Xinje XDPPro project, PLC1: XD5E-60 (software 3.8.0a 2025-04-30)

PROGRAM 梯形图

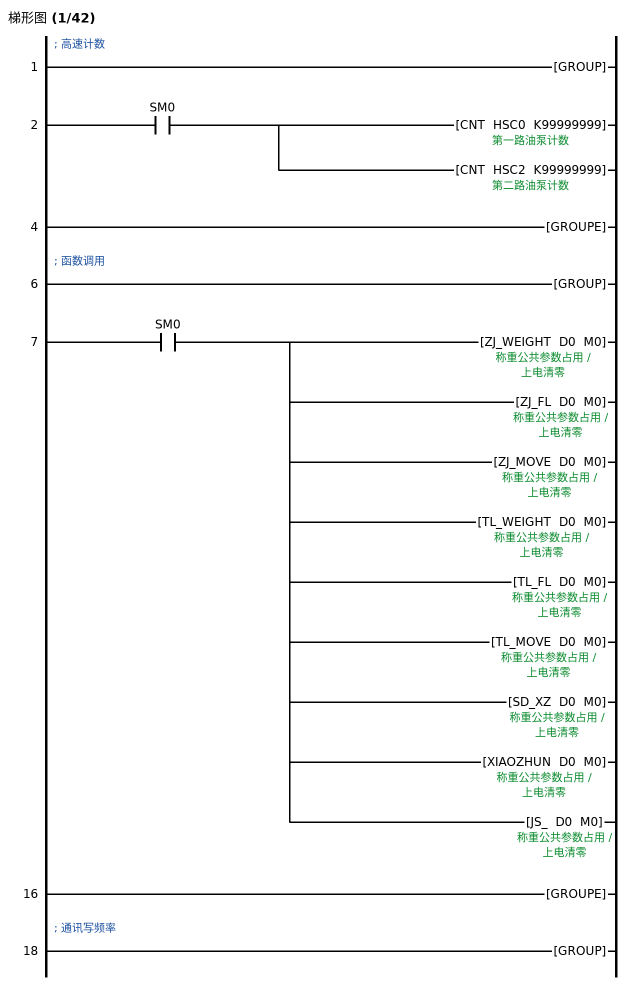
; 高速计数
GROUP
LD     SM0
CNT    HSC0 K99999999	; 第一路油泵计数
CNT    HSC2 K99999999	; 第二路油泵计数
GROUPE
; 函数调用
GROUP
LD     SM0
ZJ_WEIGHT D0 M0	; 称重公共参数占用 / 上电清零
ZJ_FL  D0 M0	; 称重公共参数占用 / 上电清零
ZJ_MOVE D0 M0	; 称重公共参数占用 / 上电清零
TL_WEIGHT D0 M0	; 称重公共参数占用 / 上电清零
TL_FL  D0 M0	; 称重公共参数占用 / 上电清零
TL_MOVE D0 M0	; 称重公共参数占用 / 上电清零
SD_XZ  D0 M0	; 称重公共参数占用 / 上电清零
XIAOZHUN D0 M0	; 称重公共参数占用 / 上电清零
JS_    D0 M0	; 称重公共参数占用 / 上电清零
GROUPE
; 通讯写频率
GROUP

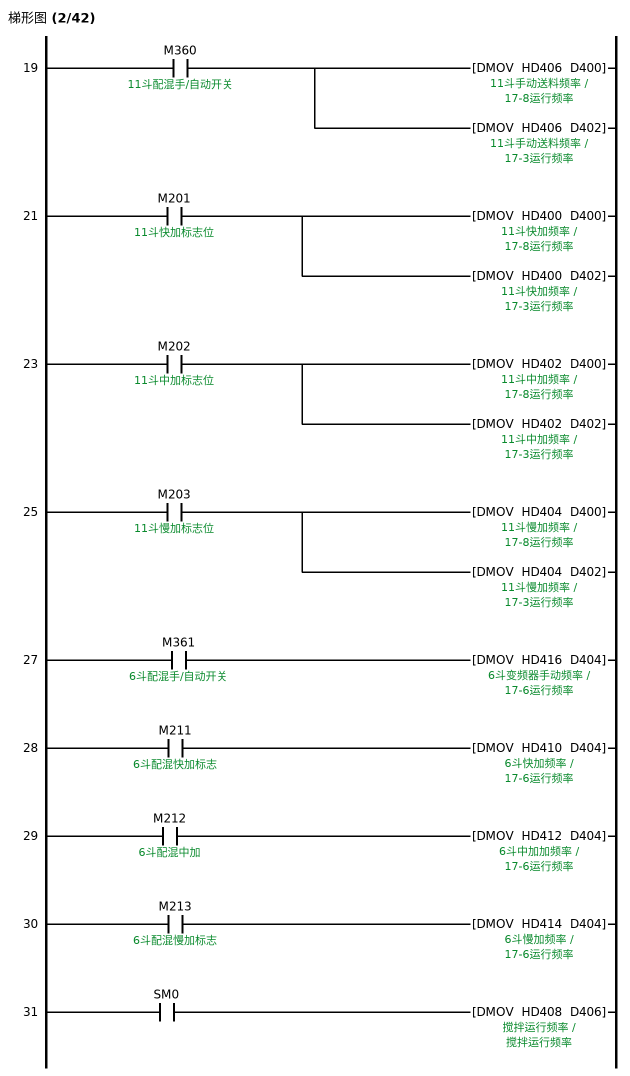
LD     M360	; 11斗配混手/自动开关
DMOV   HD406 D400	; 11斗手动送料频率 / 17-8运行频率
DMOV   HD406 D402	; 11斗手动送料频率 / 17-3运行频率
LD     M201	; 11斗快加标志位
DMOV   HD400 D400	; 11斗快加频率 / 17-8运行频率
DMOV   HD400 D402	; 11斗快加频率 / 17-3运行频率
LD     M202	; 11斗中加标志位
DMOV   HD402 D400	; 11斗中加频率 / 17-8运行频率
DMOV   HD402 D402	; 11斗中加频率 / 17-3运行频率
LD     M203	; 11斗慢加标志位
DMOV   HD404 D400	; 11斗慢加频率 / 17-8运行频率
DMOV   HD404 D402	; 11斗慢加频率 / 17-3运行频率
LD     M361	; 6斗配混手/自动开关
DMOV   HD416 D404	; 6斗变频器手动频率 / 17-6运行频率
LD     M211	; 6斗配混快加标志
DMOV   HD410 D404	; 6斗快加频率 / 17-6运行频率
LD     M212	; 6斗配混中加
DMOV   HD412 D404	; 6斗中加加频率 / 17-6运行频率
LD     M213	; 6斗配混慢加标志
DMOV   HD414 D404	; 6斗慢加频率 / 17-6运行频率
LD     SM0
DMOV   HD408 D406	; 搅拌运行频率 / 搅拌运行频率

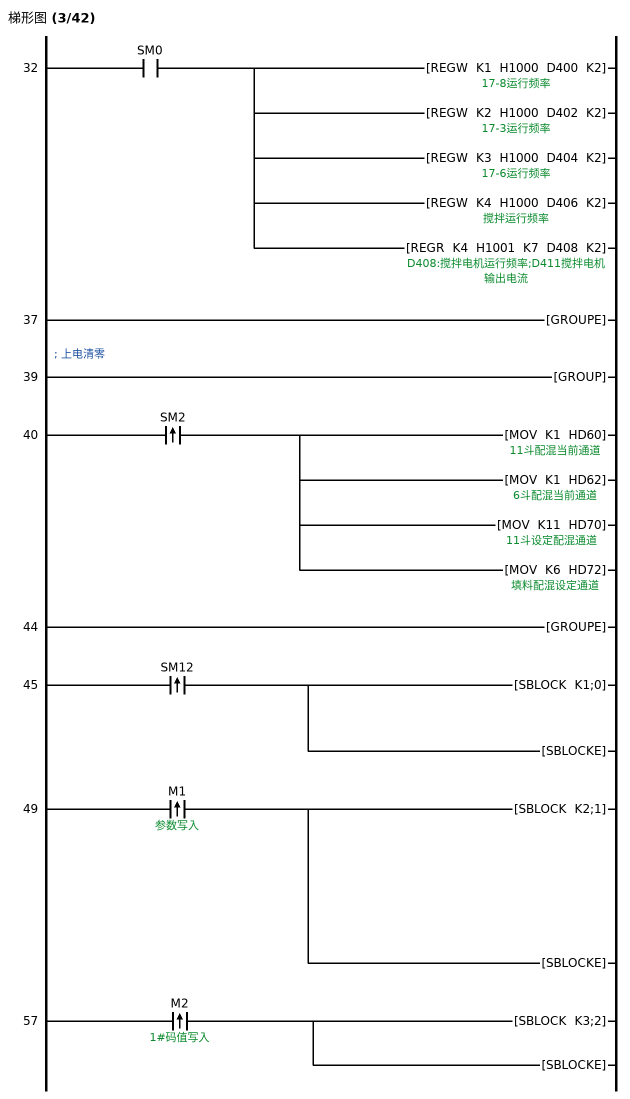
LD     SM0
REGW   K1 H1000 D400 K2	; 17-8运行频率
REGW   K2 H1000 D402 K2	; 17-3运行频率
REGW   K3 H1000 D404 K2	; 17-6运行频率
REGW   K4 H1000 D406 K2	; 搅拌运行频率
REGR   K4 H1001 K7 D408 K2	; D408:搅拌电机运行频率;D411搅拌电机输出电流
GROUPE
; 上电清零
GROUP
LDP    SM2
MOV    K1 HD60	; 11斗配混当前通道
MOV    K1 HD62	; 6斗配混当前通道
MOV    K11 HD70	; 11斗设定配混通道
MOV    K6 HD72	; 填料配混设定通道
GROUPE
LDP    SM12
SBLOCK K1;0
SBLOCKE
LDP    M1	; 参数写入
SBLOCK K2;1
SBLOCKE
LDP    M2	; 1#码值写入
SBLOCK K3;2
SBLOCKE

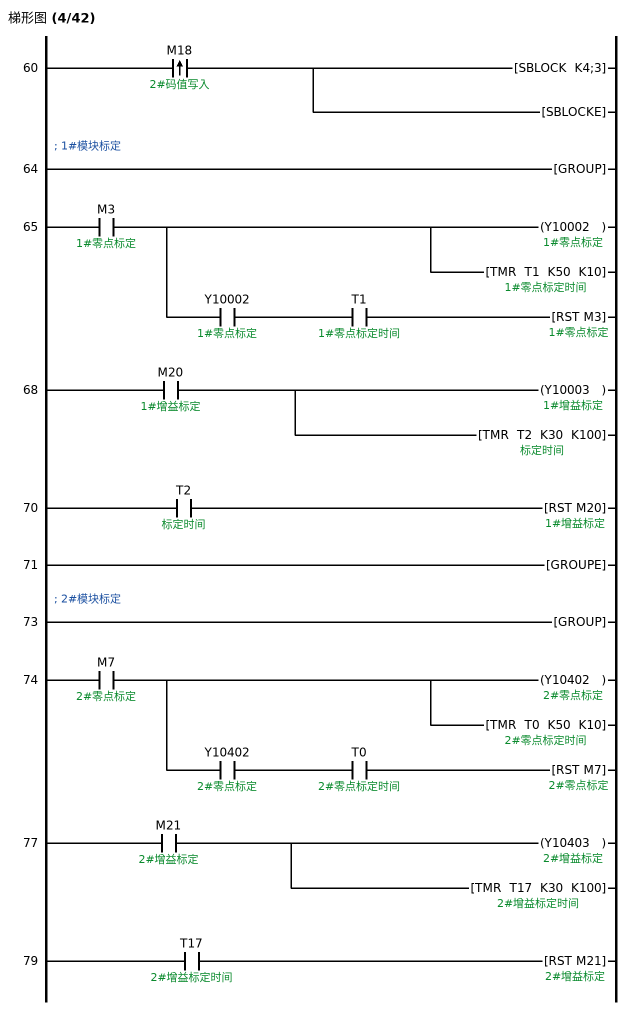
LDP    M18	; 2#码值写入
SBLOCK K4;3
SBLOCKE
; 1#模块标定
GROUP
LD     M3	; 1#零点标定
OUT    Y10002	; 1#零点标定
TMR    T1 K50 K10	; 1#零点标定时间
AND    Y10002	; 1#零点标定
AND    T1	; 1#零点标定时间
RST    M3	; 1#零点标定
LD     M20	; 1#增益标定
OUT    Y10003	; 1#增益标定
TMR    T2 K30 K100	; 标定时间
LD     T2	; 标定时间
RST    M20	; 1#增益标定
GROUPE
; 2#模块标定
GROUP
LD     M7	; 2#零点标定
OUT    Y10402	; 2#零点标定
TMR    T0 K50 K10	; 2#零点标定时间
AND    Y10402	; 2#零点标定
AND    T0	; 2#零点标定时间
RST    M7	; 2#零点标定
LD     M21	; 2#增益标定
OUT    Y10403	; 2#增益标定
TMR    T17 K30 K100	; 2#增益标定时间
LD     T17	; 2#增益标定时间
RST    M21	; 2#增益标定

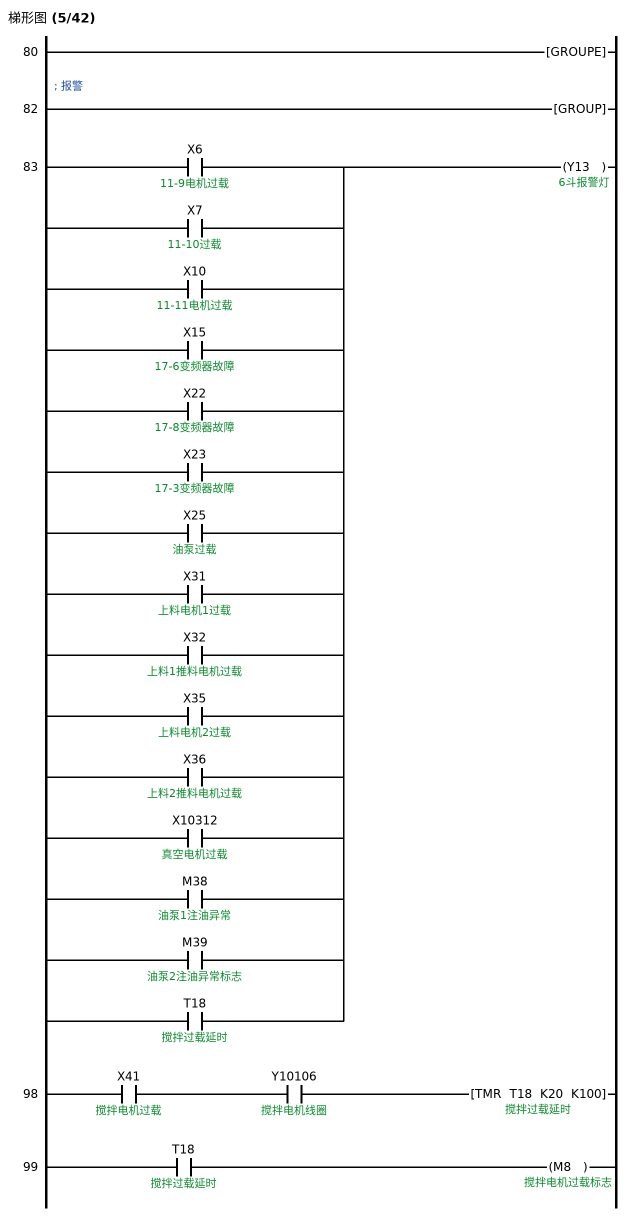
GROUPE
; 报警
GROUP
LD     X6	; 11-9电机过载
OR     X7	; 11-10过载
OR     X10	; 11-11电机过载
OR     X15	; 17-6变频器故障
OR     X22	; 17-8变频器故障
OR     X23	; 17-3变频器故障
OR     X25	; 油泵过载
OR     X31	; 上料电机1过载
OR     X32	; 上料1推料电机过载
OR     X35	; 上料电机2过载
OR     X36	; 上料2推料电机过载
OR     X10312	; 真空电机过载
OR     M38	; 油泵1注油异常
OR     M39	; 油泵2注油异常标志
OR     T18	; 搅拌过载延时
OUT    Y13	; 6斗报警灯
LD     X41	; 搅拌电机过载
AND    Y10106	; 搅拌电机线圈
TMR    T18 K20 K100	; 搅拌过载延时
LD     T18	; 搅拌过载延时
OUT    M8	; 搅拌电机过载标志

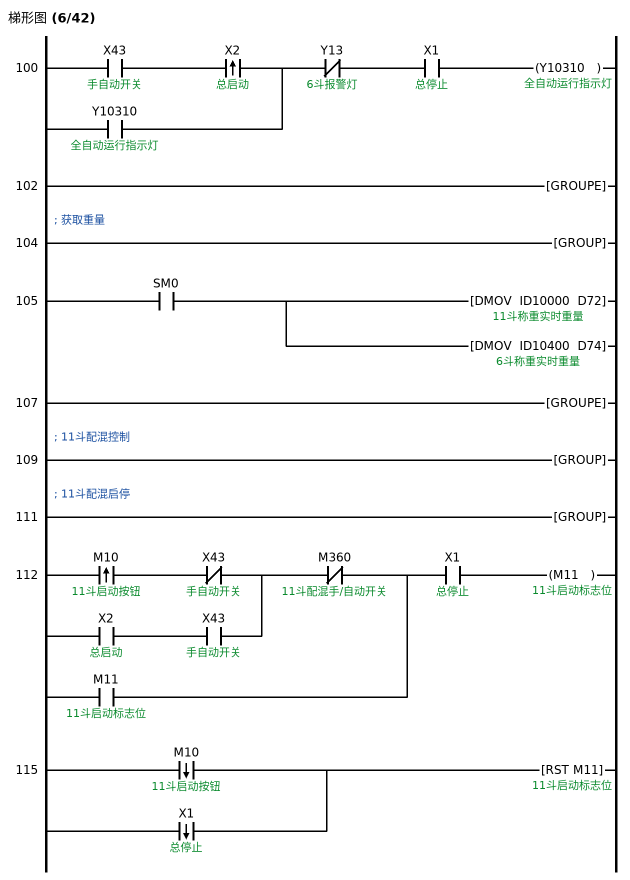
LD     X43	; 手自动开关
ANDP   X2	; 总启动
OR     Y10310	; 全自动运行指示灯
ANI    Y13	; 6斗报警灯
AND    X1	; 总停止
OUT    Y10310	; 全自动运行指示灯
GROUPE
; 获取重量
GROUP
LD     SM0
DMOV   ID10000 D72	; 11斗称重实时重量
DMOV   ID10400 D74	; 6斗称重实时重量
GROUPE
; 11斗配混控制
GROUP
; 11斗配混启停
GROUP
LDP    M10	; 11斗启动按钮
ANI    X43	; 手自动开关
LD     X2	; 总启动
AND    X43	; 手自动开关
ORB
ANI    M360	; 11斗配混手/自动开关
OR     M11	; 11斗启动标志位
AND    X1	; 总停止
OUT    M11	; 11斗启动标志位
LDF    M10	; 11斗启动按钮
ORF    X1	; 总停止
RST    M11	; 11斗启动标志位

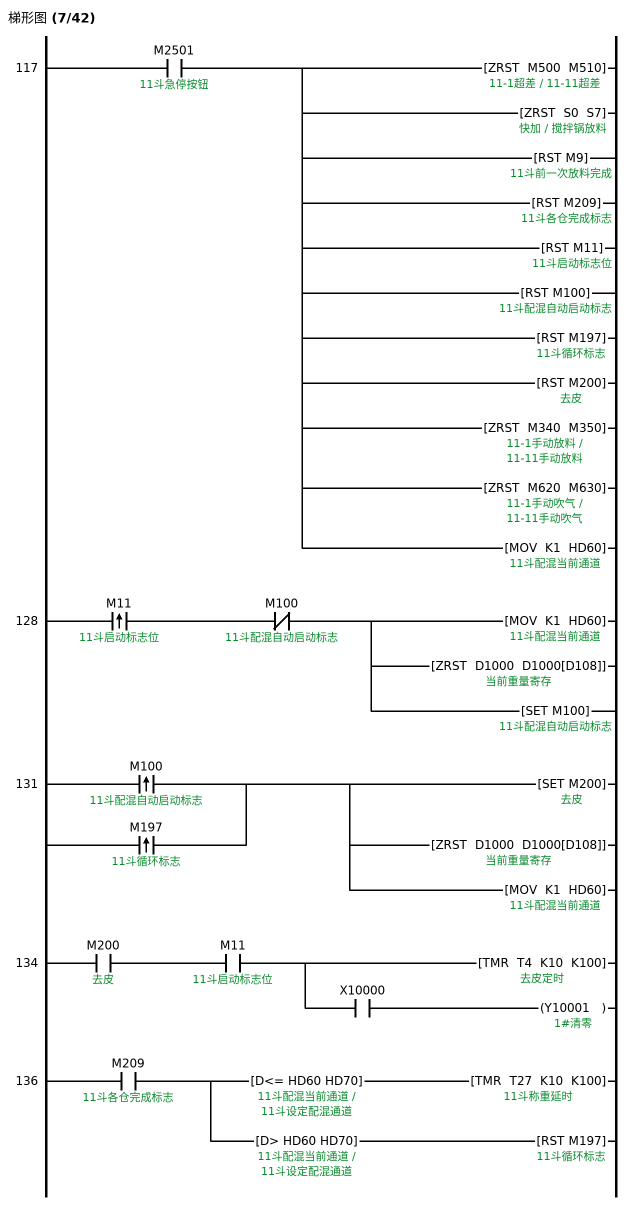
LD     M2501	; 11斗急停按钮
ZRST   M500 M510	; 11-1超差 / 11-11超差
ZRST   S0 S7	; 快加 / 搅拌锅放料
RST    M9	; 11斗前一次放料完成
RST    M209	; 11斗各仓完成标志
RST    M11	; 11斗启动标志位
RST    M100	; 11斗配混自动启动标志
RST    M197	; 11斗循环标志
RST    M200	; 去皮
ZRST   M340 M350	; 11-1手动放料 / 11-11手动放料
ZRST   M620 M630	; 11-1手动吹气 / 11-11手动吹气
MOV    K1 HD60	; 11斗配混当前通道
LDP    M11	; 11斗启动标志位
ANI    M100	; 11斗配混自动启动标志
MOV    K1 HD60	; 11斗配混当前通道
ZRST   D1000 D1000[D108]	; 当前重量寄存
SET    M100	; 11斗配混自动启动标志
LDP    M100	; 11斗配混自动启动标志
ORP    M197	; 11斗循环标志
SET    M200	; 去皮
ZRST   D1000 D1000[D108]	; 当前重量寄存
MOV    K1 HD60	; 11斗配混当前通道
LD     M200	; 去皮
AND    M11	; 11斗启动标志位
TMR    T4 K10 K100	; 去皮定时
AND    X10000
OUT    Y10001	; 1#清零
LD     M209	; 11斗各仓完成标志
MPS
DAND<= HD60 HD70	; 11斗配混当前通道 / 11斗设定配混通道
TMR    T27 K10 K100	; 11斗称重延时
MPP
DAND>  HD60 HD70	; 11斗配混当前通道 / 11斗设定配混通道
RST    M197	; 11斗循环标志

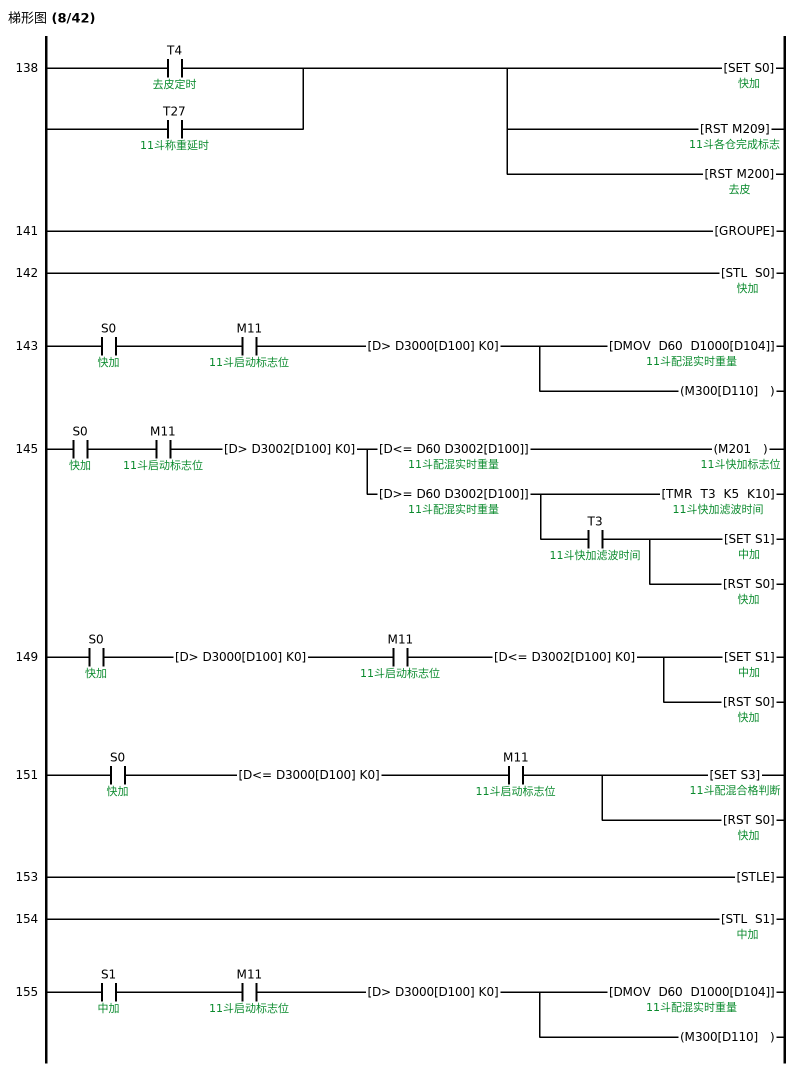
LD     T4	; 去皮定时
OR     T27	; 11斗称重延时
SET    S0	; 快加
RST    M209	; 11斗各仓完成标志
RST    M200	; 去皮
GROUPE
STL    S0	; 快加
LD     S0	; 快加
AND    M11	; 11斗启动标志位
DAND>  D3000[D100] K0
DMOV   D60 D1000[D104]	; 11斗配混实时重量
OUT    M300[D110]
LD     S0	; 快加
AND    M11	; 11斗启动标志位
DAND>  D3002[D100] K0
MPS
DAND<= D60 D3002[D100]	; 11斗配混实时重量
OUT    M201	; 11斗快加标志位
MPP
DAND>= D60 D3002[D100]	; 11斗配混实时重量
TMR    T3 K5 K10	; 11斗快加滤波时间
AND    T3	; 11斗快加滤波时间
SET    S1	; 中加
RST    S0	; 快加
LD     S0	; 快加
DAND>  D3000[D100] K0
AND    M11	; 11斗启动标志位
DAND<= D3002[D100] K0
SET    S1	; 中加
RST    S0	; 快加
LD     S0	; 快加
DAND<= D3000[D100] K0
AND    M11	; 11斗启动标志位
SET    S3	; 11斗配混合格判断
RST    S0	; 快加
STLE
STL    S1	; 中加
LD     S1	; 中加
AND    M11	; 11斗启动标志位
DAND>  D3000[D100] K0
DMOV   D60 D1000[D104]	; 11斗配混实时重量
OUT    M300[D110]

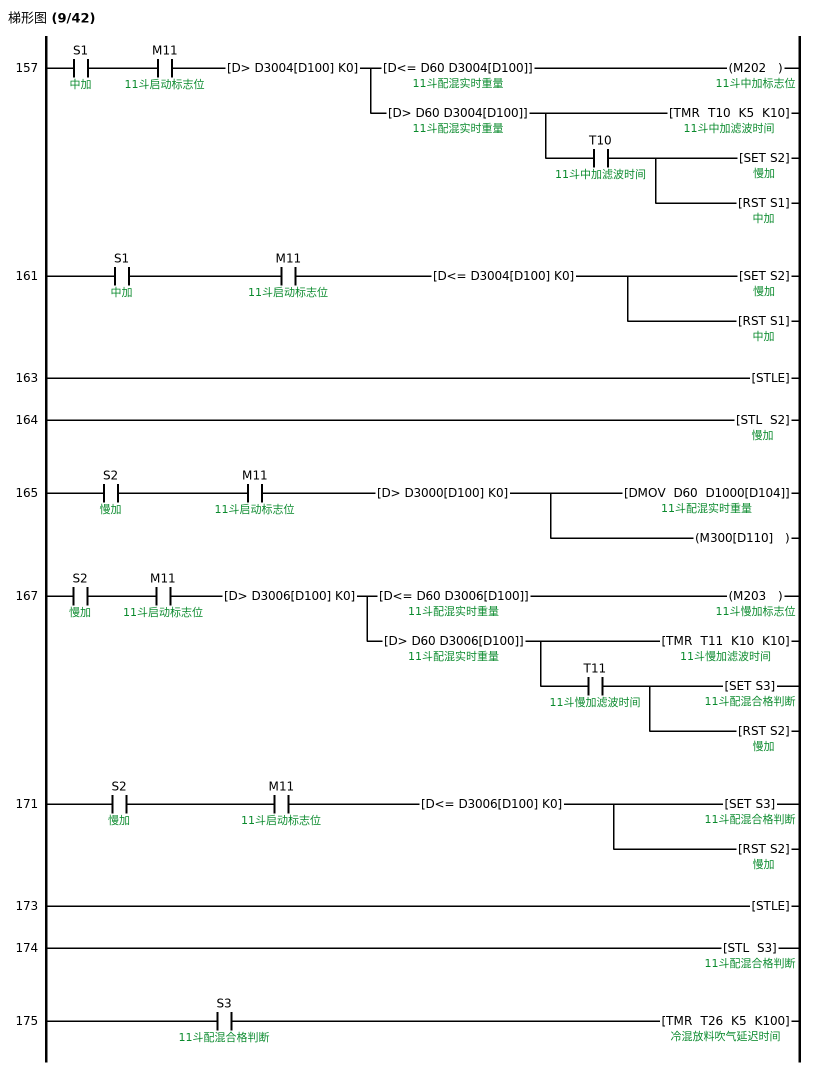
LD     S1	; 中加
AND    M11	; 11斗启动标志位
DAND>  D3004[D100] K0
MPS
DAND<= D60 D3004[D100]	; 11斗配混实时重量
OUT    M202	; 11斗中加标志位
MPP
DAND>  D60 D3004[D100]	; 11斗配混实时重量
TMR    T10 K5 K10	; 11斗中加滤波时间
AND    T10	; 11斗中加滤波时间
SET    S2	; 慢加
RST    S1	; 中加
LD     S1	; 中加
AND    M11	; 11斗启动标志位
DAND<= D3004[D100] K0
SET    S2	; 慢加
RST    S1	; 中加
STLE
STL    S2	; 慢加
LD     S2	; 慢加
AND    M11	; 11斗启动标志位
DAND>  D3000[D100] K0
DMOV   D60 D1000[D104]	; 11斗配混实时重量
OUT    M300[D110]
LD     S2	; 慢加
AND    M11	; 11斗启动标志位
DAND>  D3006[D100] K0
MPS
DAND<= D60 D3006[D100]	; 11斗配混实时重量
OUT    M203	; 11斗慢加标志位
MPP
DAND>  D60 D3006[D100]	; 11斗配混实时重量
TMR    T11 K10 K10	; 11斗慢加滤波时间
AND    T11	; 11斗慢加滤波时间
SET    S3	; 11斗配混合格判断
RST    S2	; 慢加
LD     S2	; 慢加
AND    M11	; 11斗启动标志位
DAND<= D3006[D100] K0
SET    S3	; 11斗配混合格判断
RST    S2	; 慢加
STLE
STL    S3	; 11斗配混合格判断
LD     S3	; 11斗配混合格判断
TMR    T26 K5 K100	; 冷混放料吹气延迟时间

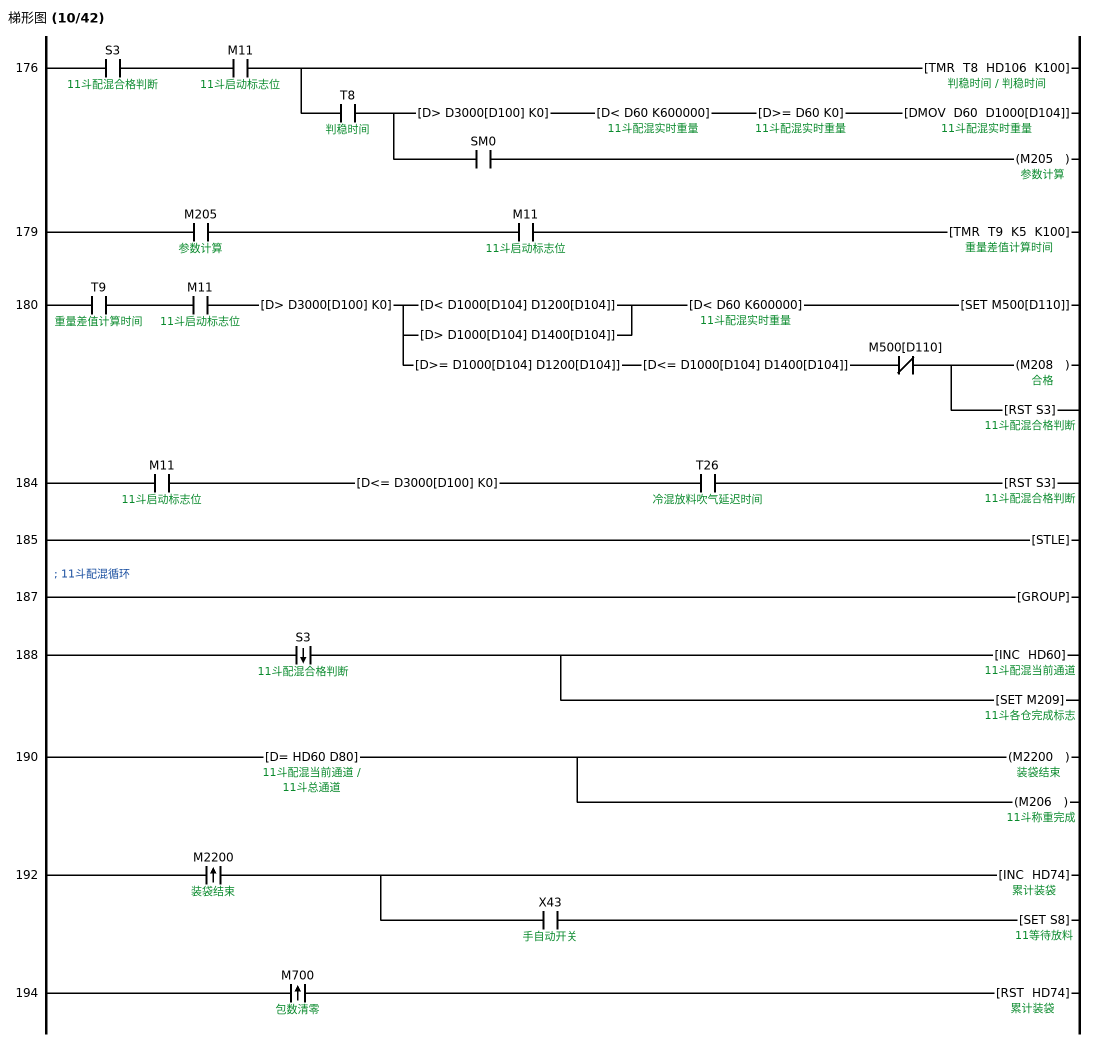
LD     S3	; 11斗配混合格判断
AND    M11	; 11斗启动标志位
TMR    T8 HD106 K100	; 判稳时间 / 判稳时间
AND    T8	; 判稳时间
MPS
DAND>  D3000[D100] K0
DAND<  D60 K600000	; 11斗配混实时重量
DAND>= D60 K0	; 11斗配混实时重量
DMOV   D60 D1000[D104]	; 11斗配混实时重量
MPP
AND    SM0
OUT    M205	; 参数计算
LD     M205	; 参数计算
AND    M11	; 11斗启动标志位
TMR    T9 K5 K100	; 重量差值计算时间
LD     T9	; 重量差值计算时间
AND    M11	; 11斗启动标志位
DAND>  D3000[D100] K0
MPS
DLD<   D1000[D104] D1200[D104]
DOR>   D1000[D104] D1400[D104]
ANB
DAND<  D60 K600000	; 11斗配混实时重量
SET    M500[D110]
MPP
DAND>= D1000[D104] D1200[D104]
DAND<= D1000[D104] D1400[D104]
ANI    M500[D110]
OUT    M208	; 合格
RST    S3	; 11斗配混合格判断
LD     M11	; 11斗启动标志位
DAND<= D3000[D100] K0
AND    T26	; 冷混放料吹气延迟时间
RST    S3	; 11斗配混合格判断
STLE
; 11斗配混循环
GROUP
LDF    S3	; 11斗配混合格判断
INC    HD60	; 11斗配混当前通道
SET    M209	; 11斗各仓完成标志
DLD=   HD60 D80	; 11斗配混当前通道 / 11斗总通道
OUT    M2200	; 装袋结束
OUT    M206	; 11斗称重完成
LDP    M2200	; 装袋结束
INC    HD74	; 累计装袋
AND    X43	; 手自动开关
SET    S8	; 11等待放料
LDP    M700	; 包数清零
RST    HD74	; 累计装袋

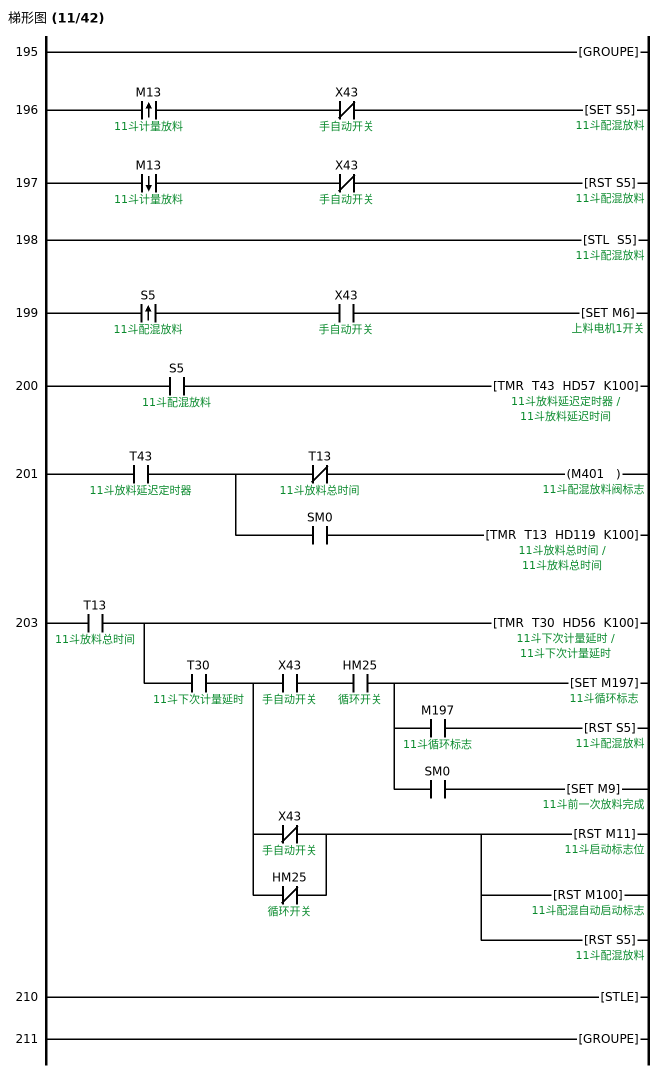
GROUPE
LDP    M13	; 11斗计量放料
ANI    X43	; 手自动开关
SET    S5	; 11斗配混放料
LDF    M13	; 11斗计量放料
ANI    X43	; 手自动开关
RST    S5	; 11斗配混放料
STL    S5	; 11斗配混放料
LDP    S5	; 11斗配混放料
AND    X43	; 手自动开关
SET    M6	; 上料电机1开关
LD     S5	; 11斗配混放料
TMR    T43 HD57 K100	; 11斗放料延迟定时器 / 11斗放料延迟时间
LD     T43	; 11斗放料延迟定时器
MPS
ANI    T13	; 11斗放料总时间
OUT    M401	; 11斗配混放料阀标志
MPP
AND    SM0
TMR    T13 HD119 K100	; 11斗放料总时间 / 11斗放料总时间
LD     T13	; 11斗放料总时间
TMR    T30 HD56 K100	; 11斗下次计量延时 / 11斗下次计量延时
AND    T30	; 11斗下次计量延时
MPS
AND    X43	; 手自动开关
AND    HM25	; 循环开关
SET    M197	; 11斗循环标志
MPS
AND    M197	; 11斗循环标志
RST    S5	; 11斗配混放料
MPP
AND    SM0
SET    M9	; 11斗前一次放料完成
MPP
LDI    X43	; 手自动开关
ORI    HM25	; 循环开关
ANB
RST    M11	; 11斗启动标志位
RST    M100	; 11斗配混自动启动标志
RST    S5	; 11斗配混放料
STLE
GROUPE

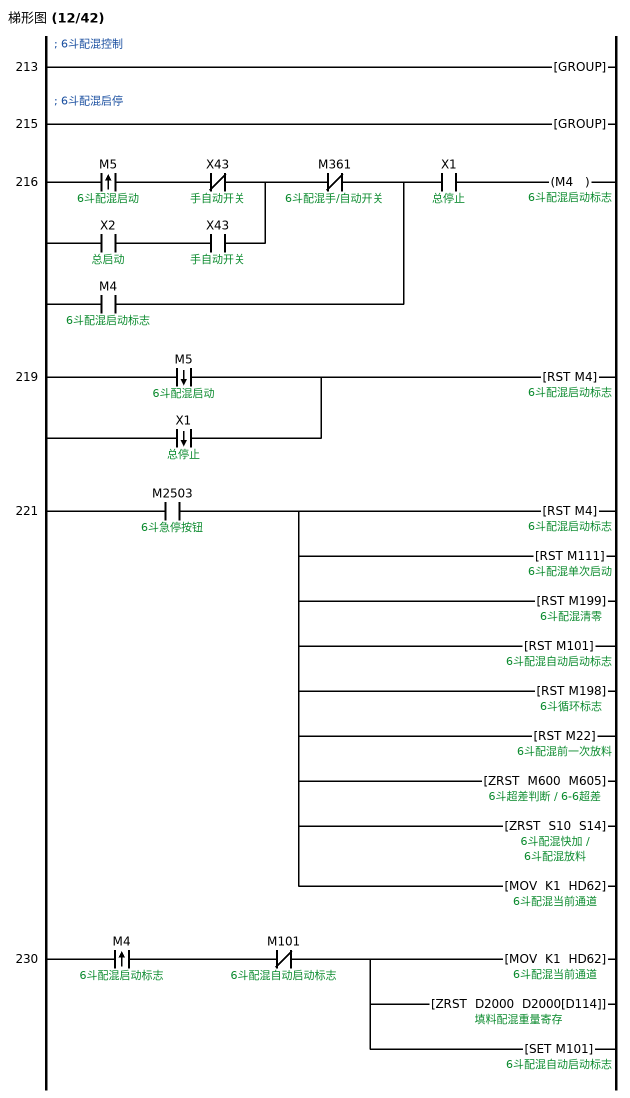
; 6斗配混控制
GROUP
; 6斗配混启停
GROUP
LDP    M5	; 6斗配混启动
ANI    X43	; 手自动开关
LD     X2	; 总启动
AND    X43	; 手自动开关
ORB
ANI    M361	; 6斗配混手/自动开关
OR     M4	; 6斗配混启动标志
AND    X1	; 总停止
OUT    M4	; 6斗配混启动标志
LDF    M5	; 6斗配混启动
ORF    X1	; 总停止
RST    M4	; 6斗配混启动标志
LD     M2503	; 6斗急停按钮
RST    M4	; 6斗配混启动标志
RST    M111	; 6斗配混单次启动
RST    M199	; 6斗配混清零
RST    M101	; 6斗配混自动启动标志
RST    M198	; 6斗循环标志
RST    M22	; 6斗配混前一次放料
ZRST   M600 M605	; 6斗超差判断 / 6-6超差
ZRST   S10 S14	; 6斗配混快加 / 6斗配混放料
MOV    K1 HD62	; 6斗配混当前通道
LDP    M4	; 6斗配混启动标志
ANI    M101	; 6斗配混自动启动标志
MOV    K1 HD62	; 6斗配混当前通道
ZRST   D2000 D2000[D114]	; 填料配混重量寄存
SET    M101	; 6斗配混自动启动标志

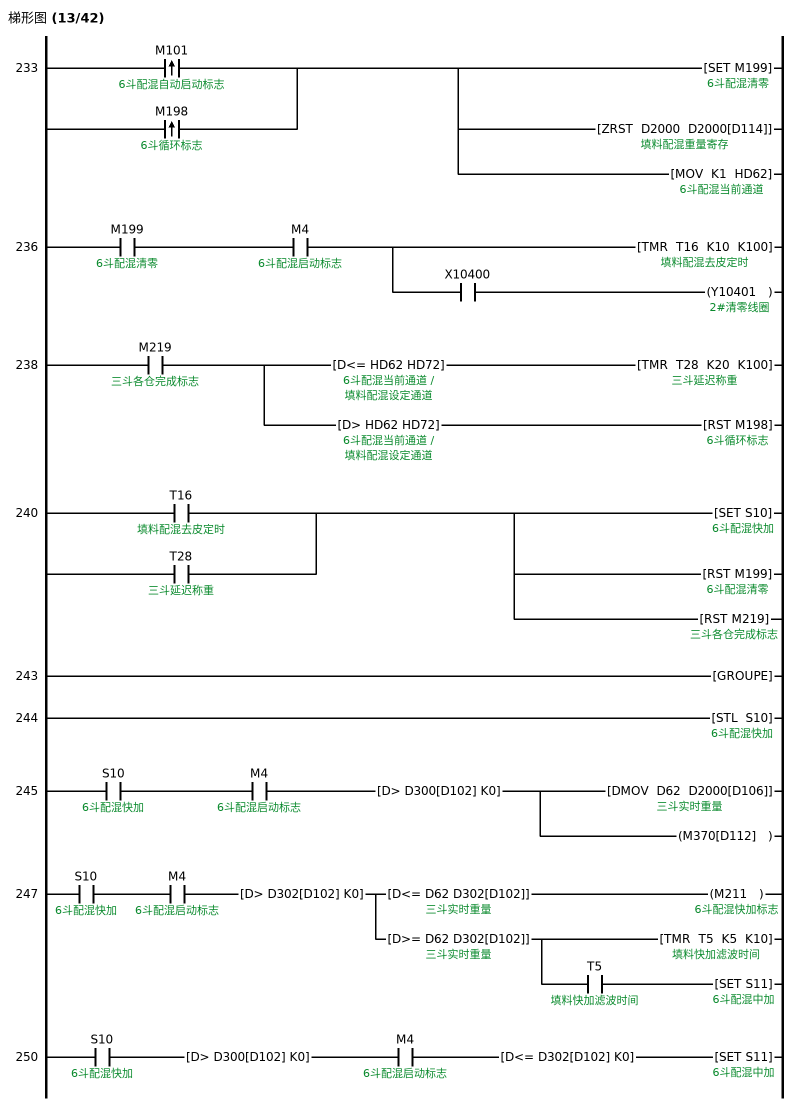
LDP    M101	; 6斗配混自动启动标志
ORP    M198	; 6斗循环标志
SET    M199	; 6斗配混清零
ZRST   D2000 D2000[D114]	; 填料配混重量寄存
MOV    K1 HD62	; 6斗配混当前通道
LD     M199	; 6斗配混清零
AND    M4	; 6斗配混启动标志
TMR    T16 K10 K100	; 填料配混去皮定时
AND    X10400
OUT    Y10401	; 2#清零线圈
LD     M219	; 三斗各仓完成标志
MPS
DAND<= HD62 HD72	; 6斗配混当前通道 / 填料配混设定通道
TMR    T28 K20 K100	; 三斗延迟称重
MPP
DAND>  HD62 HD72	; 6斗配混当前通道 / 填料配混设定通道
RST    M198	; 6斗循环标志
LD     T16	; 填料配混去皮定时
OR     T28	; 三斗延迟称重
SET    S10	; 6斗配混快加
RST    M199	; 6斗配混清零
RST    M219	; 三斗各仓完成标志
GROUPE
STL    S10	; 6斗配混快加
LD     S10	; 6斗配混快加
AND    M4	; 6斗配混启动标志
DAND>  D300[D102] K0
DMOV   D62 D2000[D106]	; 三斗实时重量
OUT    M370[D112]
LD     S10	; 6斗配混快加
AND    M4	; 6斗配混启动标志
DAND>  D302[D102] K0
MPS
DAND<= D62 D302[D102]	; 三斗实时重量
OUT    M211	; 6斗配混快加标志
MPP
DAND>= D62 D302[D102]	; 三斗实时重量
TMR    T5 K5 K10	; 填料快加滤波时间
AND    T5	; 填料快加滤波时间
SET    S11	; 6斗配混中加
LD     S10	; 6斗配混快加
DAND>  D300[D102] K0
AND    M4	; 6斗配混启动标志
DAND<= D302[D102] K0
SET    S11	; 6斗配混中加

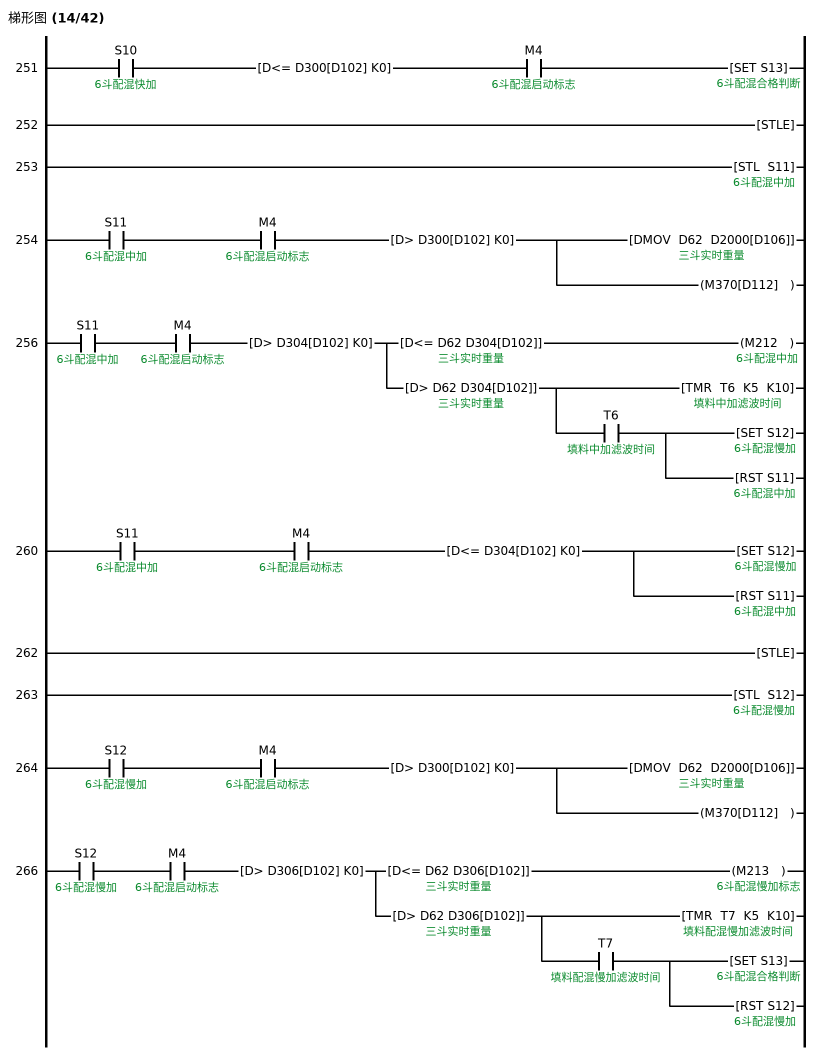
LD     S10	; 6斗配混快加
DAND<= D300[D102] K0
AND    M4	; 6斗配混启动标志
SET    S13	; 6斗配混合格判断
STLE
STL    S11	; 6斗配混中加
LD     S11	; 6斗配混中加
AND    M4	; 6斗配混启动标志
DAND>  D300[D102] K0
DMOV   D62 D2000[D106]	; 三斗实时重量
OUT    M370[D112]
LD     S11	; 6斗配混中加
AND    M4	; 6斗配混启动标志
DAND>  D304[D102] K0
MPS
DAND<= D62 D304[D102]	; 三斗实时重量
OUT    M212	; 6斗配混中加
MPP
DAND>  D62 D304[D102]	; 三斗实时重量
TMR    T6 K5 K10	; 填料中加滤波时间
AND    T6	; 填料中加滤波时间
SET    S12	; 6斗配混慢加
RST    S11	; 6斗配混中加
LD     S11	; 6斗配混中加
AND    M4	; 6斗配混启动标志
DAND<= D304[D102] K0
SET    S12	; 6斗配混慢加
RST    S11	; 6斗配混中加
STLE
STL    S12	; 6斗配混慢加
LD     S12	; 6斗配混慢加
AND    M4	; 6斗配混启动标志
DAND>  D300[D102] K0
DMOV   D62 D2000[D106]	; 三斗实时重量
OUT    M370[D112]
LD     S12	; 6斗配混慢加
AND    M4	; 6斗配混启动标志
DAND>  D306[D102] K0
MPS
DAND<= D62 D306[D102]	; 三斗实时重量
OUT    M213	; 6斗配混慢加标志
MPP
DAND>  D62 D306[D102]	; 三斗实时重量
TMR    T7 K5 K10	; 填料配混慢加滤波时间
AND    T7	; 填料配混慢加滤波时间
SET    S13	; 6斗配混合格判断
RST    S12	; 6斗配混慢加

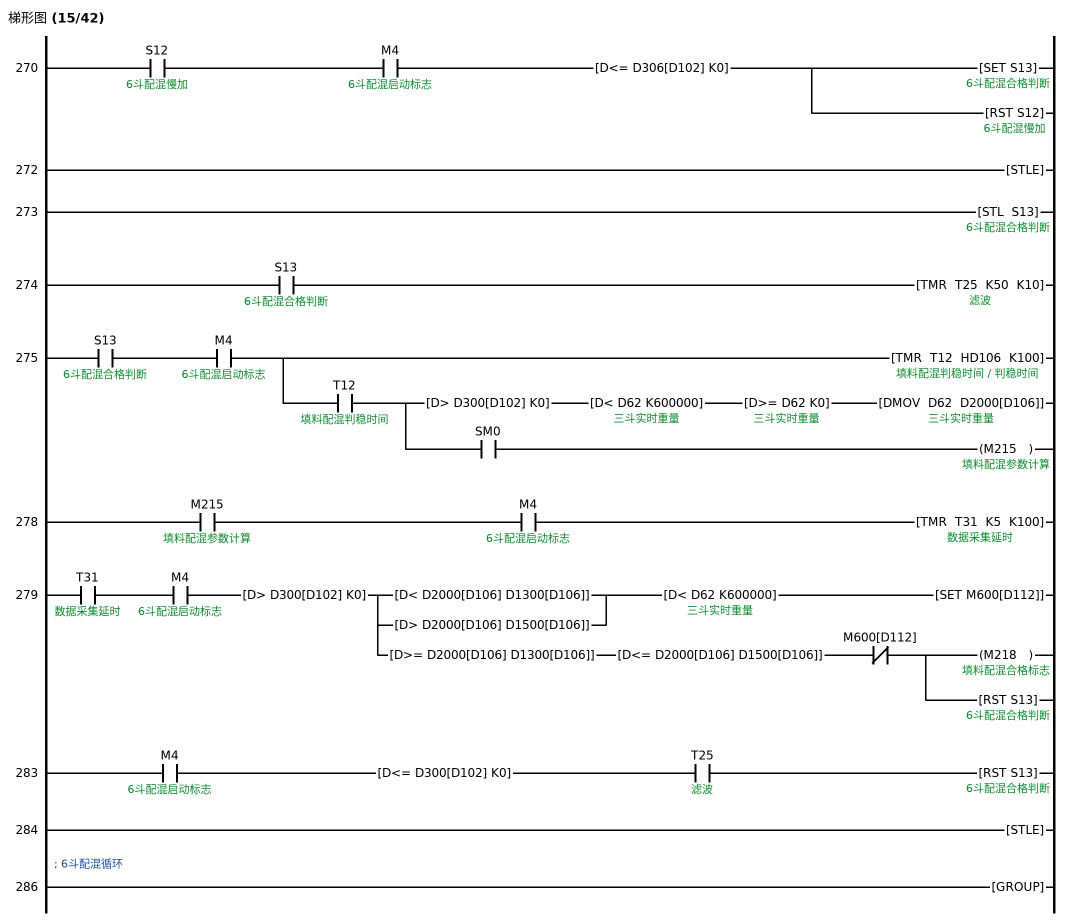
LD     S12	; 6斗配混慢加
AND    M4	; 6斗配混启动标志
DAND<= D306[D102] K0
SET    S13	; 6斗配混合格判断
RST    S12	; 6斗配混慢加
STLE
STL    S13	; 6斗配混合格判断
LD     S13	; 6斗配混合格判断
TMR    T25 K50 K10	; 滤波
LD     S13	; 6斗配混合格判断
AND    M4	; 6斗配混启动标志
TMR    T12 HD106 K100	; 填料配混判稳时间 / 判稳时间
AND    T12	; 填料配混判稳时间
MPS
DAND>  D300[D102] K0
DAND<  D62 K600000	; 三斗实时重量
DAND>= D62 K0	; 三斗实时重量
DMOV   D62 D2000[D106]	; 三斗实时重量
MPP
AND    SM0
OUT    M215	; 填料配混参数计算
LD     M215	; 填料配混参数计算
AND    M4	; 6斗配混启动标志
TMR    T31 K5 K100	; 数据采集延时
LD     T31	; 数据采集延时
AND    M4	; 6斗配混启动标志
DAND>  D300[D102] K0
MPS
DLD<   D2000[D106] D1300[D106]
DOR>   D2000[D106] D1500[D106]
ANB
DAND<  D62 K600000	; 三斗实时重量
SET    M600[D112]
MPP
DAND>= D2000[D106] D1300[D106]
DAND<= D2000[D106] D1500[D106]
ANI    M600[D112]
OUT    M218	; 填料配混合格标志
RST    S13	; 6斗配混合格判断
LD     M4	; 6斗配混启动标志
DAND<= D300[D102] K0
AND    T25	; 滤波
RST    S13	; 6斗配混合格判断
STLE
; 6斗配混循环
GROUP

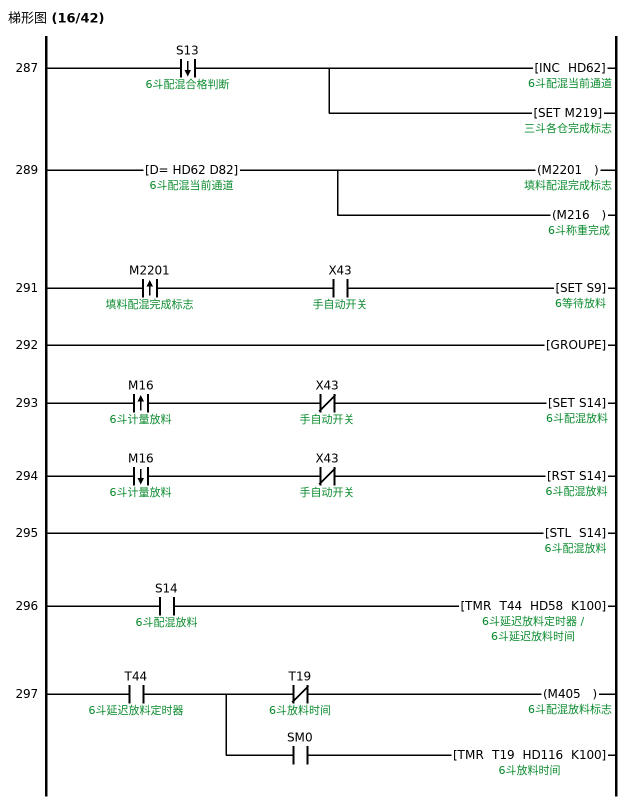
LDF    S13	; 6斗配混合格判断
INC    HD62	; 6斗配混当前通道
SET    M219	; 三斗各仓完成标志
DLD=   HD62 D82	; 6斗配混当前通道
OUT    M2201	; 填料配混完成标志
OUT    M216	; 6斗称重完成
LDP    M2201	; 填料配混完成标志
AND    X43	; 手自动开关
SET    S9	; 6等待放料
GROUPE
LDP    M16	; 6斗计量放料
ANI    X43	; 手自动开关
SET    S14	; 6斗配混放料
LDF    M16	; 6斗计量放料
ANI    X43	; 手自动开关
RST    S14	; 6斗配混放料
STL    S14	; 6斗配混放料
LD     S14	; 6斗配混放料
TMR    T44 HD58 K100	; 6斗延迟放料定时器 / 6斗延迟放料时间
LD     T44	; 6斗延迟放料定时器
MPS
ANI    T19	; 6斗放料时间
OUT    M405	; 6斗配混放料标志
MPP
AND    SM0
TMR    T19 HD116 K100	; 6斗放料时间

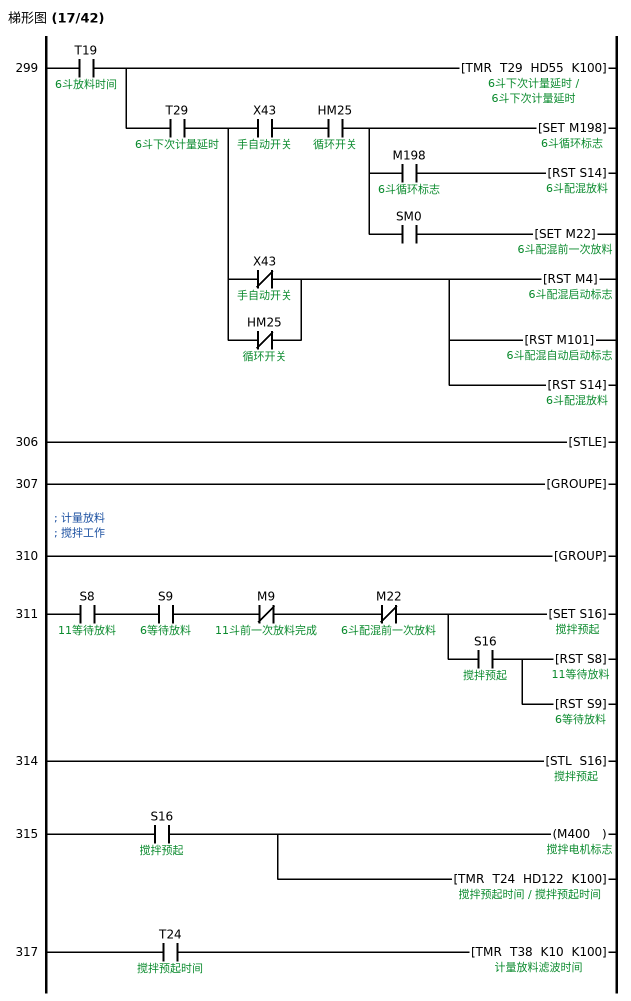
LD     T19	; 6斗放料时间
TMR    T29 HD55 K100	; 6斗下次计量延时 / 6斗下次计量延时
AND    T29	; 6斗下次计量延时
MPS
AND    X43	; 手自动开关
AND    HM25	; 循环开关
SET    M198	; 6斗循环标志
MPS
AND    M198	; 6斗循环标志
RST    S14	; 6斗配混放料
MPP
AND    SM0
SET    M22	; 6斗配混前一次放料
MPP
LDI    X43	; 手自动开关
ORI    HM25	; 循环开关
ANB
RST    M4	; 6斗配混启动标志
RST    M101	; 6斗配混自动启动标志
RST    S14	; 6斗配混放料
STLE
GROUPE
; 计量放料
; 搅拌工作
GROUP
LD     S8	; 11等待放料
AND    S9	; 6等待放料
ANI    M9	; 11斗前一次放料完成
ANI    M22	; 6斗配混前一次放料
SET    S16	; 搅拌预起
AND    S16	; 搅拌预起
RST    S8	; 11等待放料
RST    S9	; 6等待放料
STL    S16	; 搅拌预起
LD     S16	; 搅拌预起
OUT    M400	; 搅拌电机标志
TMR    T24 HD122 K100	; 搅拌预起时间 / 搅拌预起时间
LD     T24	; 搅拌预起时间
TMR    T38 K10 K100	; 计量放料滤波时间

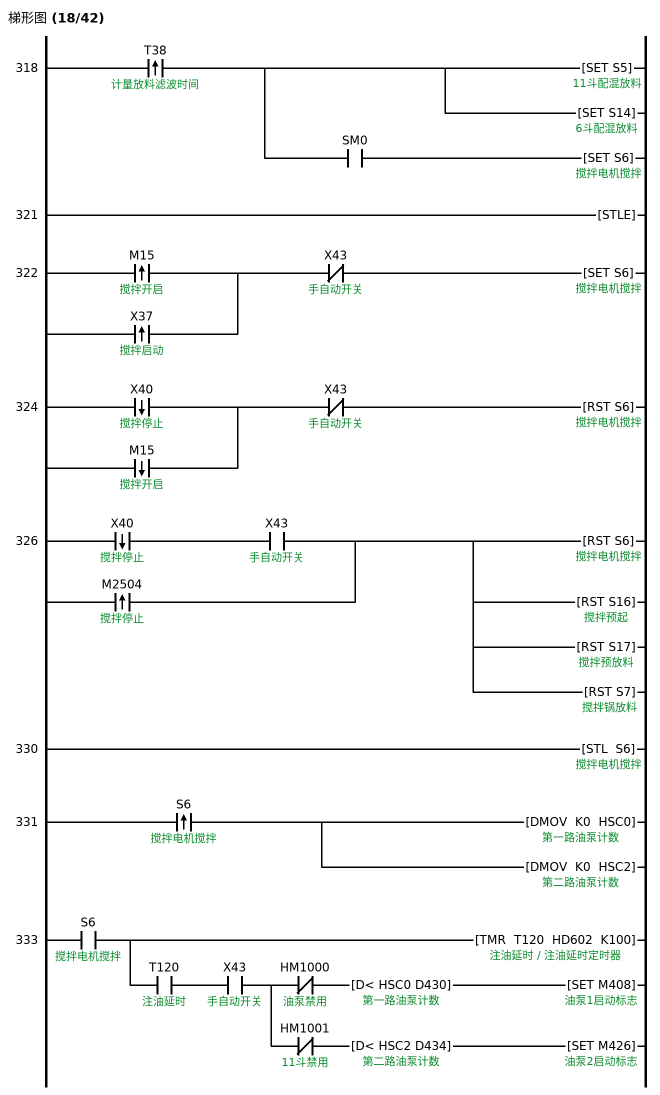
LDP    T38	; 计量放料滤波时间
SET    S5	; 11斗配混放料
SET    S14	; 6斗配混放料
AND    SM0
SET    S6	; 搅拌电机搅拌
STLE
LDP    M15	; 搅拌开启
ORP    X37	; 搅拌启动
ANI    X43	; 手自动开关
SET    S6	; 搅拌电机搅拌
LDF    X40	; 搅拌停止
ORF    M15	; 搅拌开启
ANI    X43	; 手自动开关
RST    S6	; 搅拌电机搅拌
LDF    X40	; 搅拌停止
AND    X43	; 手自动开关
ORP    M2504	; 搅拌停止
RST    S6	; 搅拌电机搅拌
RST    S16	; 搅拌预起
RST    S17	; 搅拌预放料
RST    S7	; 搅拌锅放料
STL    S6	; 搅拌电机搅拌
LDP    S6	; 搅拌电机搅拌
DMOV   K0 HSC0	; 第一路油泵计数
DMOV   K0 HSC2	; 第二路油泵计数
LD     S6	; 搅拌电机搅拌
TMR    T120 HD602 K100	; 注油延时 / 注油延时定时器
AND    T120	; 注油延时
AND    X43	; 手自动开关
MPS
ANI    HM1000	; 油泵禁用
DAND<  HSC0 D430	; 第一路油泵计数
SET    M408	; 油泵1启动标志
MPP
ANI    HM1001	; 11斗禁用
DAND<  HSC2 D434	; 第二路油泵计数
SET    M426	; 油泵2启动标志

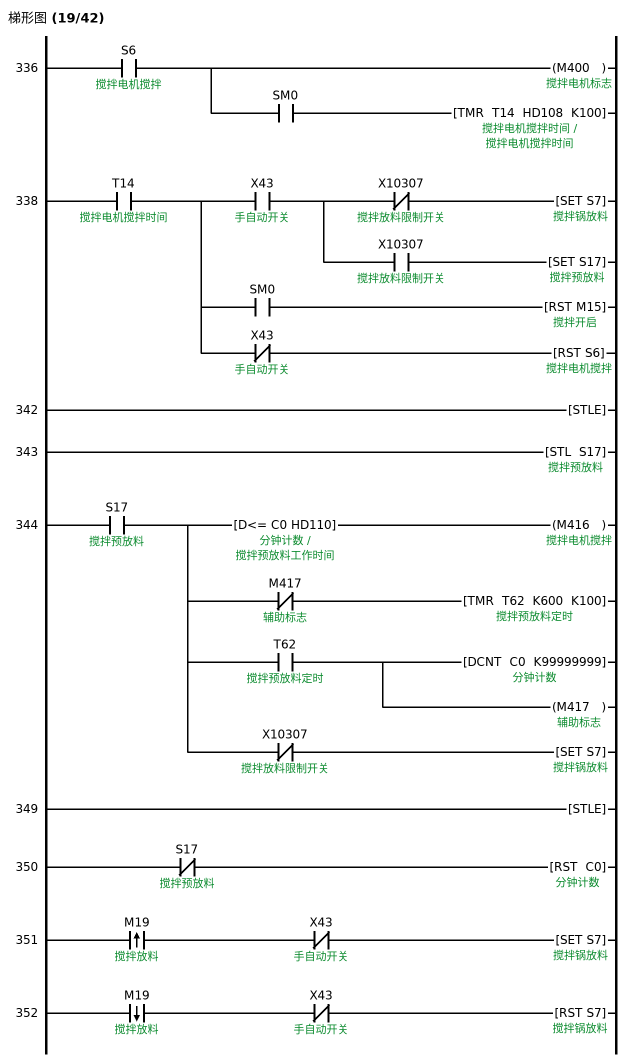
LD     S6	; 搅拌电机搅拌
OUT    M400	; 搅拌电机标志
AND    SM0
TMR    T14 HD108 K100	; 搅拌电机搅拌时间 / 搅拌电机搅拌时间
LD     T14	; 搅拌电机搅拌时间
MPS
AND    X43	; 手自动开关
MPS
ANI    X10307	; 搅拌放料限制开关
SET    S7	; 搅拌锅放料
MPP
AND    X10307	; 搅拌放料限制开关
SET    S17	; 搅拌预放料
MRD
AND    SM0
RST    M15	; 搅拌开启
MPP
ANI    X43	; 手自动开关
RST    S6	; 搅拌电机搅拌
STLE
STL    S17	; 搅拌预放料
LD     S17	; 搅拌预放料
MPS
DAND<= C0 HD110	; 分钟计数 / 搅拌预放料工作时间
OUT    M416	; 搅拌电机搅拌
MRD
ANI    M417	; 辅助标志
TMR    T62 K600 K100	; 搅拌预放料定时
MRD
AND    T62	; 搅拌预放料定时
DCNT   C0 K99999999	; 分钟计数
OUT    M417	; 辅助标志
MPP
ANI    X10307	; 搅拌放料限制开关
SET    S7	; 搅拌锅放料
STLE
LDI    S17	; 搅拌预放料
RST    C0	; 分钟计数
LDP    M19	; 搅拌放料
ANI    X43	; 手自动开关
SET    S7	; 搅拌锅放料
LDF    M19	; 搅拌放料
ANI    X43	; 手自动开关
RST    S7	; 搅拌锅放料

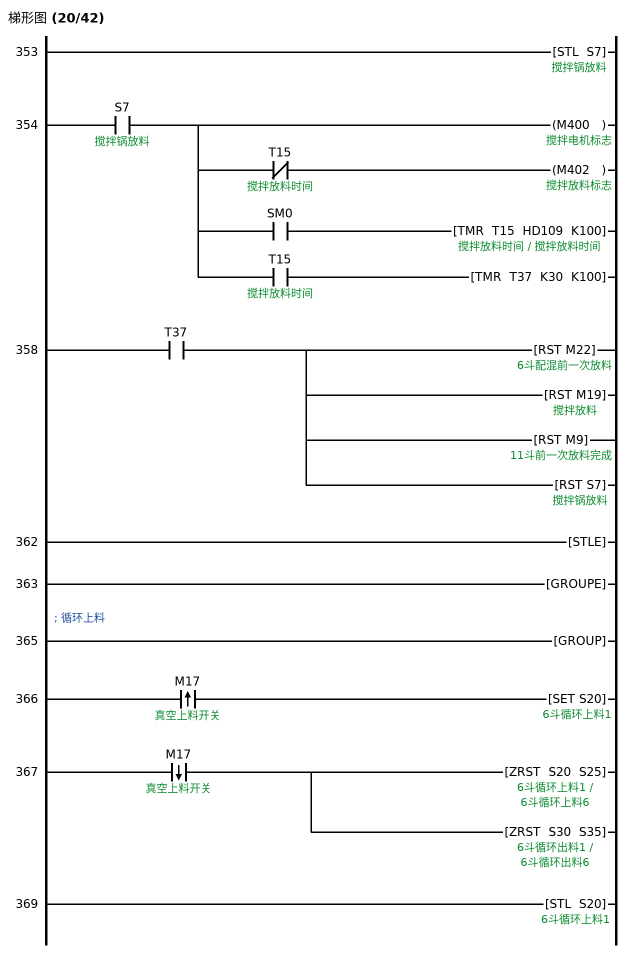
STL    S7	; 搅拌锅放料
LD     S7	; 搅拌锅放料
OUT    M400	; 搅拌电机标志
MPS
ANI    T15	; 搅拌放料时间
OUT    M402	; 搅拌放料标志
MRD
AND    SM0
TMR    T15 HD109 K100	; 搅拌放料时间 / 搅拌放料时间
MPP
AND    T15	; 搅拌放料时间
TMR    T37 K30 K100
LD     T37
RST    M22	; 6斗配混前一次放料
RST    M19	; 搅拌放料
RST    M9	; 11斗前一次放料完成
RST    S7	; 搅拌锅放料
STLE
GROUPE
; 循环上料
GROUP
LDP    M17	; 真空上料开关
SET    S20	; 6斗循环上料1
LDF    M17	; 真空上料开关
ZRST   S20 S25	; 6斗循环上料1 / 6斗循环上料6
ZRST   S30 S35	; 6斗循环出料1 / 6斗循环出料6
STL    S20	; 6斗循环上料1

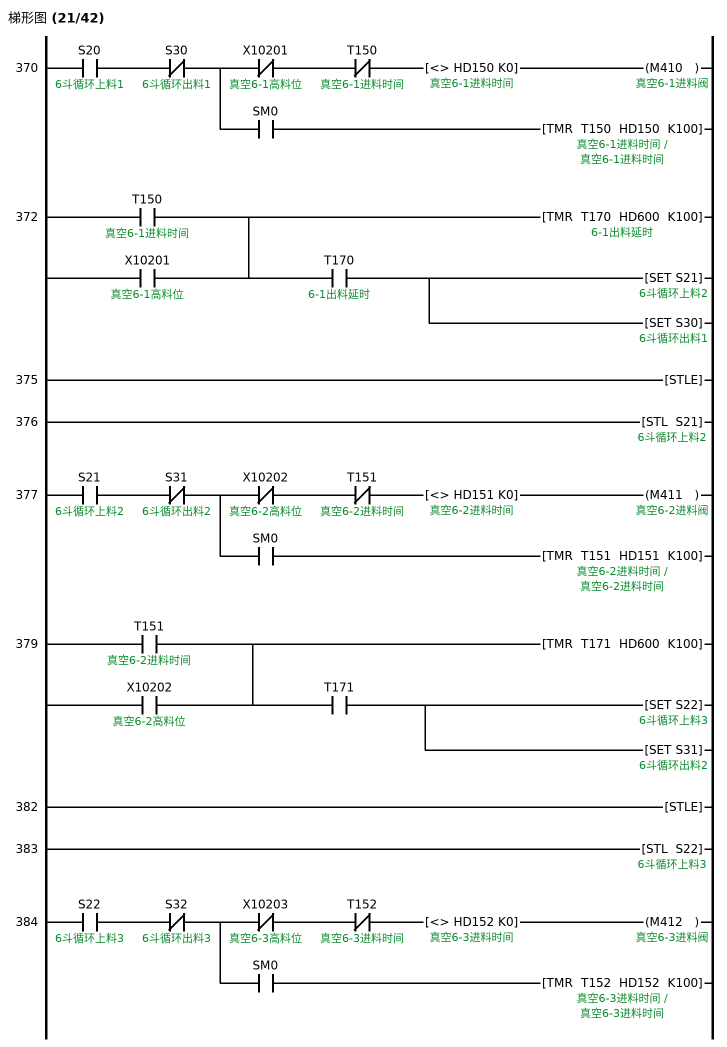
LD     S20	; 6斗循环上料1
ANI    S30	; 6斗循环出料1
MPS
ANI    X10201	; 真空6-1高料位
ANI    T150	; 真空6-1进料时间
AND<>  HD150 K0	; 真空6-1进料时间
OUT    M410	; 真空6-1进料阀
MPP
AND    SM0
TMR    T150 HD150 K100	; 真空6-1进料时间 / 真空6-1进料时间
LD     T150	; 真空6-1进料时间
OR     X10201	; 真空6-1高料位
TMR    T170 HD600 K100	; 6-1出料延时
AND    T170	; 6-1出料延时
SET    S21	; 6斗循环上料2
SET    S30	; 6斗循环出料1
STLE
STL    S21	; 6斗循环上料2
LD     S21	; 6斗循环上料2
ANI    S31	; 6斗循环出料2
MPS
ANI    X10202	; 真空6-2高料位
ANI    T151	; 真空6-2进料时间
AND<>  HD151 K0	; 真空6-2进料时间
OUT    M411	; 真空6-2进料阀
MPP
AND    SM0
TMR    T151 HD151 K100	; 真空6-2进料时间 / 真空6-2进料时间
LD     T151	; 真空6-2进料时间
OR     X10202	; 真空6-2高料位
TMR    T171 HD600 K100
AND    T171
SET    S22	; 6斗循环上料3
SET    S31	; 6斗循环出料2
STLE
STL    S22	; 6斗循环上料3
LD     S22	; 6斗循环上料3
ANI    S32	; 6斗循环出料3
MPS
ANI    X10203	; 真空6-3高料位
ANI    T152	; 真空6-3进料时间
AND<>  HD152 K0	; 真空6-3进料时间
OUT    M412	; 真空6-3进料阀
MPP
AND    SM0
TMR    T152 HD152 K100	; 真空6-3进料时间 / 真空6-3进料时间

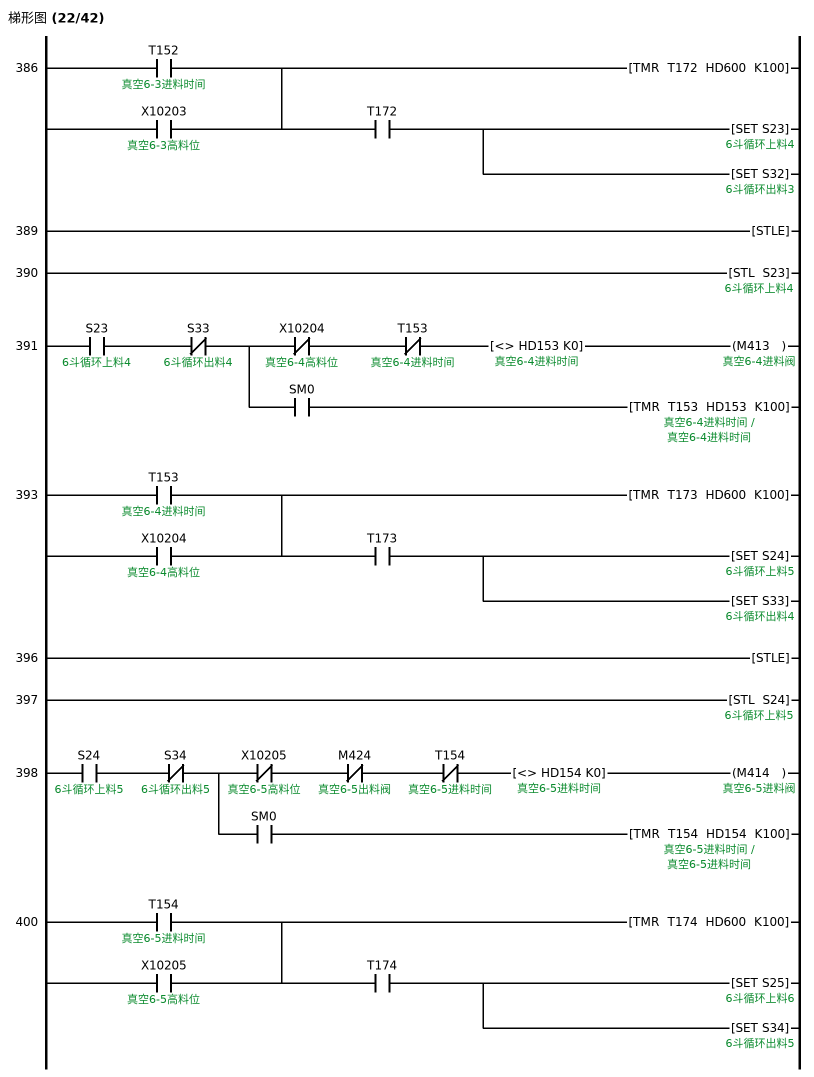
LD     T152	; 真空6-3进料时间
OR     X10203	; 真空6-3高料位
TMR    T172 HD600 K100
AND    T172
SET    S23	; 6斗循环上料4
SET    S32	; 6斗循环出料3
STLE
STL    S23	; 6斗循环上料4
LD     S23	; 6斗循环上料4
ANI    S33	; 6斗循环出料4
MPS
ANI    X10204	; 真空6-4高料位
ANI    T153	; 真空6-4进料时间
AND<>  HD153 K0	; 真空6-4进料时间
OUT    M413	; 真空6-4进料阀
MPP
AND    SM0
TMR    T153 HD153 K100	; 真空6-4进料时间 / 真空6-4进料时间
LD     T153	; 真空6-4进料时间
OR     X10204	; 真空6-4高料位
TMR    T173 HD600 K100
AND    T173
SET    S24	; 6斗循环上料5
SET    S33	; 6斗循环出料4
STLE
STL    S24	; 6斗循环上料5
LD     S24	; 6斗循环上料5
ANI    S34	; 6斗循环出料5
MPS
ANI    X10205	; 真空6-5高料位
ANI    M424	; 真空6-5出料阀
ANI    T154	; 真空6-5进料时间
AND<>  HD154 K0	; 真空6-5进料时间
OUT    M414	; 真空6-5进料阀
MPP
AND    SM0
TMR    T154 HD154 K100	; 真空6-5进料时间 / 真空6-5进料时间
LD     T154	; 真空6-5进料时间
OR     X10205	; 真空6-5高料位
TMR    T174 HD600 K100
AND    T174
SET    S25	; 6斗循环上料6
SET    S34	; 6斗循环出料5

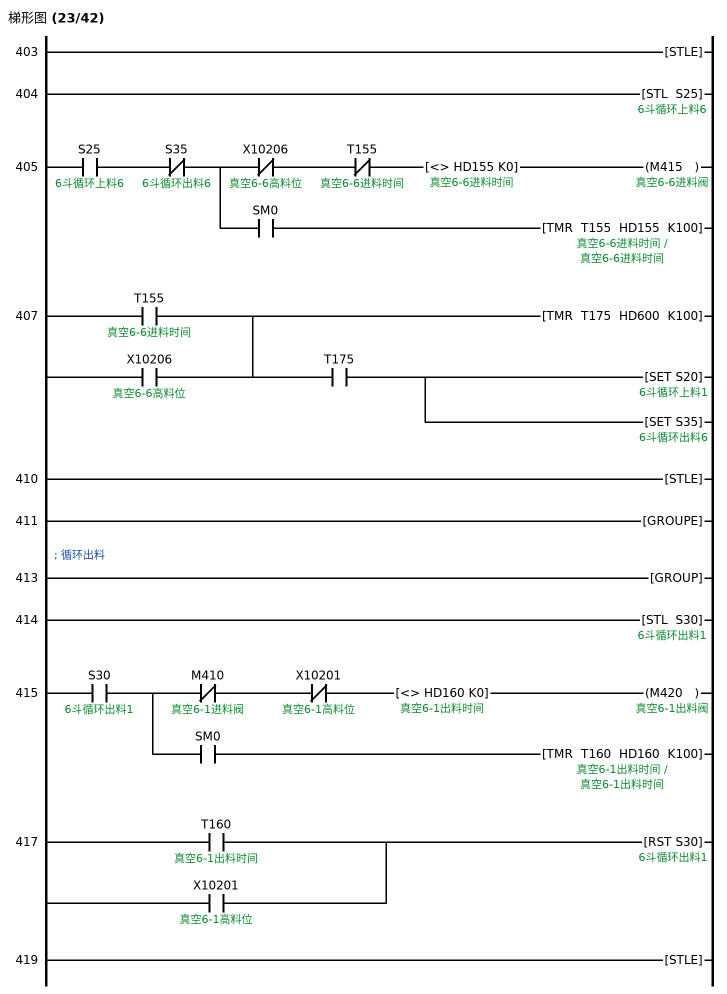
STLE
STL    S25	; 6斗循环上料6
LD     S25	; 6斗循环上料6
ANI    S35	; 6斗循环出料6
MPS
ANI    X10206	; 真空6-6高料位
ANI    T155	; 真空6-6进料时间
AND<>  HD155 K0	; 真空6-6进料时间
OUT    M415	; 真空6-6进料阀
MPP
AND    SM0
TMR    T155 HD155 K100	; 真空6-6进料时间 / 真空6-6进料时间
LD     T155	; 真空6-6进料时间
OR     X10206	; 真空6-6高料位
TMR    T175 HD600 K100
AND    T175
SET    S20	; 6斗循环上料1
SET    S35	; 6斗循环出料6
STLE
GROUPE
; 循环出料
GROUP
STL    S30	; 6斗循环出料1
LD     S30	; 6斗循环出料1
MPS
ANI    M410	; 真空6-1进料阀
ANI    X10201	; 真空6-1高料位
AND<>  HD160 K0	; 真空6-1出料时间
OUT    M420	; 真空6-1出料阀
MPP
AND    SM0
TMR    T160 HD160 K100	; 真空6-1出料时间 / 真空6-1出料时间
LD     T160	; 真空6-1出料时间
OR     X10201	; 真空6-1高料位
RST    S30	; 6斗循环出料1
STLE

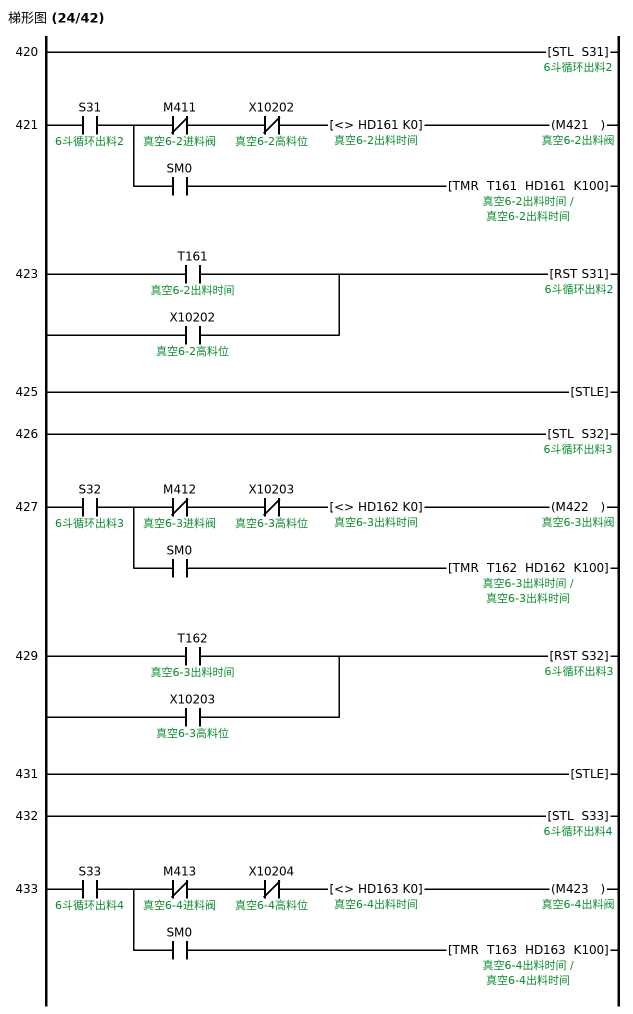
STL    S31	; 6斗循环出料2
LD     S31	; 6斗循环出料2
MPS
ANI    M411	; 真空6-2进料阀
ANI    X10202	; 真空6-2高料位
AND<>  HD161 K0	; 真空6-2出料时间
OUT    M421	; 真空6-2出料阀
MPP
AND    SM0
TMR    T161 HD161 K100	; 真空6-2出料时间 / 真空6-2出料时间
LD     T161	; 真空6-2出料时间
OR     X10202	; 真空6-2高料位
RST    S31	; 6斗循环出料2
STLE
STL    S32	; 6斗循环出料3
LD     S32	; 6斗循环出料3
MPS
ANI    M412	; 真空6-3进料阀
ANI    X10203	; 真空6-3高料位
AND<>  HD162 K0	; 真空6-3出料时间
OUT    M422	; 真空6-3出料阀
MPP
AND    SM0
TMR    T162 HD162 K100	; 真空6-3出料时间 / 真空6-3出料时间
LD     T162	; 真空6-3出料时间
OR     X10203	; 真空6-3高料位
RST    S32	; 6斗循环出料3
STLE
STL    S33	; 6斗循环出料4
LD     S33	; 6斗循环出料4
MPS
ANI    M413	; 真空6-4进料阀
ANI    X10204	; 真空6-4高料位
AND<>  HD163 K0	; 真空6-4出料时间
OUT    M423	; 真空6-4出料阀
MPP
AND    SM0
TMR    T163 HD163 K100	; 真空6-4出料时间 / 真空6-4出料时间

